FUNCTION_BLOCK ABSTRACT FB_SaMElement EXTENDS FB_BaseComponent IMPLEMENTS ITF_SaMElement
VAR
	bActive						: BOOL;				//informacja czy dany element jest aktywny 
	bIsEnabled					: BOOL;				//informacje czy dany element jest włączony
//	refstDaneSITP				: REFERENCE TO ST_SITP_DaneElementu;
END_VAR
VAR PERSISTENT
	ltWorkTime					: LTIME;				//czas pracy w danym stanie - trybie
END_VAR

METHOD PUBLIC IncrementTime
VAR_INPUT
	tInterval				: TIME := T#100MS;
END_VAR
THIS^.ltWorkTime			:= THIS^.ltWorkTime + TO_LTIME (tInterval);
END_METHOD

METHOD PUBLIC InvokeStateForTopElement : BOOL
VAR_INPUT
	itfTopElement		: ITF_BaseSaMStateMethod;
END_VAR
END_METHOD

METHOD PUBLIC IsActive : BOOL
VAR_INPUT
END_VAR
IsActive			:= THIS^.bActive;
END_METHOD

(*			
	EVERDE sp. z o.o.
	Rafał Osajda		03.11.2025		TC 4024.66
	Zwraca czy element jest właczony w systemie
*)
METHOD PUBLIC IsEnabled : BOOL
VAR_INPUT
END_VAR
IsEnabled			:= THIS^.bIsEnabled;
END_METHOD

METHOD PUBLIC ResetTime
VAR_INPUT
END_VAR
THIS^.ltWorkTime		:= LTIME#0MS;
END_METHOD

(*			
	EVERDE sp. z o.o.
	Rafał Osajda		03.11.2025		TC 4024.66
	Ustawia czy dane element jest aktywny
*)
METHOD PUBLIC SetActive
VAR_INPUT
	bIN			: BOOL;
END_VAR
THIS^.bActive	:= bIN;
END_METHOD

(*			
	EVERDE sp. z o.o.
	Rafał Osajda		03.11.2025		TC 4024.66
	Ustawie czy element jest włączony w systemie
*)
METHOD PUBLIC SetEnabled
VAR_INPUT
	bIN			: BOOL;
END_VAR
THIS^.bIsEnabled		:= bIN;
END_METHOD

END_FUNCTION_BLOCK

(* stored: Version 1.1.0.1
   POU FB_SaMElement: Id {03aaa14d-d8d1-0ccd-22ca-7daa896b0e09}, SpecialFunc None
   Method IncrementTime: Id {304bcff5-f12b-0ac9-38cb-f597f33e927e}
   Method InvokeStateForTopElement: Id {6567004d-543a-0afb-18b9-4317e3330f74}
   Method IsActive: Id {0737c9dc-d560-0e62-3c1f-3b7ef8ae10dc}
   Method IsEnabled: Id {cda05f82-8147-0995-0f93-35b325b598b2}
   Method ResetTime: Id {99320a18-e3c5-086e-3eea-75bf7272336f}
   Method SetActive: Id {335a6819-5ef9-0396-0548-e2fbc0cd5a33}
   Method SetEnabled: Id {d993afe0-6068-084d-0e12-cadc7945aa48} *)
